// TIA Portal project "StaiteMixare" (V15.1)

(* hardware
DEVICE "S71500/ET200MP station_1"  S7-1500 station
   slot 0: "Rail_0"  Rack  6ES7 590-1***0-0AA0
   slot 1: "PLC_1"  CPU 1513-1 PN  6ES7 513-1AL02-0AB0  V2.6
      slot 3: "CPU display_1"  6ES7591-1AA00-0AA0
DEVICE "HMI_1"  KTP900 Basic PN
   slot 0: "HMI_1"  KTP900 Basic PN  6AV2 123-2JB03-0AX0  15.1.0.0
   slot 1: "HMI_RT_1"  KTP900 Basic PN  6AV2 123-2JB03-0AX0  15.1.0.0
   slot 5: "HMI_1.IE_CP_1"  PROFINET Interface  15.0.1.0
      slot 1: "PROFINET Interface_1"  PROFINET Interface
         slot 1: "Port_1"  Port
*)

// ===== PLC "PLC_1"  CPU 1513-1 PN =====

VAR_GLOBAL   // PLC tag table "Default tag table"
   "Clock_Byte" AT %MB0 : Byte;
   "Clock_10Hz" AT %M0.0 : Bool;
   "Clock_5Hz" AT %M0.1 : Bool;
   "Clock_2.5Hz" AT %M0.2 : Bool;
   "Clock_2Hz" AT %M0.3 : Bool;
   "Clock_1.25Hz" AT %M0.4 : Bool;
   "Clock_1Hz" AT %M0.5 : Bool;
   "Clock_0.625Hz" AT %M0.6 : Bool;
   "Clock_0.5Hz" AT %M0.7 : Bool;
END_VAR

DATA_BLOCK "Alarme"   // DB1
{ S7_Optimized_Access := 'TRUE' }
VERSION : 0.1
   VAR
      alarme_gather : Word;
      alarme_vect : Array[0..15] of Bool;
   END_VAR
BEGIN
END_DATA_BLOCK

DATA_BLOCK "Avarii"   // DB2
{ S7_Optimized_Access := 'TRUE' }
VERSION : 0.1
   VAR
      ESD : Bool;
      esd_btn : Bool;
      reset_esd : Bool;
      avarie_mixer : Bool;
      avarie_container : Bool;
      avarie_solutie_A : Bool;
      avarie_solutie_B : Bool;
      avarie_generala : Bool;
      reset_avarie_generala : Bool;
   END_VAR
BEGIN
END_DATA_BLOCK

DATA_BLOCK "Mixer_DB"   // DB3
{ S7_Optimized_Access := 'TRUE' }
VERSION : 0.1
   VAR
      durata_mixer : Time;
      timp_trecut_secunde : Time;
      timp_elapsed : Time;
      mixer_pornit : Bool;
      plecare_stea : Bool;
      plecare_triunghi : Bool;
      btn_pornire : Bool;
   END_VAR
BEGIN
END_DATA_BLOCK

DATA_BLOCK "Container_DB"   // DB4
{ S7_Optimized_Access := 'TRUE' }
VERSION : 0.1
   VAR
      recipient : Bool := true;
      valva_golire_deschisa : Bool;
      pornire_golire : Bool;
      btn_pornire : Bool;
      debit_total : UInt := 100;
      debit_curent : UInt;
      debit_recipient : UInt := 5;
   END_VAR
BEGIN
END_DATA_BLOCK

DATA_BLOCK "Solutie_A_DB"   // DB5
{ S7_Optimized_Access := 'TRUE' }
VERSION : 0.1
   VAR
      debit_solutie : UInt := 60;
      debit_aux : UInt;
      debit_de_umplut : UInt := 20;
      debit_curent : UInt;
      indice : UInt := 1;
      btn_reumplere : Bool;
      capacitate_necesara : Bool;
      btn_pornire : Bool;
      pornite_golire : Bool;
   END_VAR
BEGIN
END_DATA_BLOCK

DATA_BLOCK "Solutie_B_DB"   // DB6
{ S7_Optimized_Access := 'TRUE' }
VERSION : 0.1
   VAR
      debit_solutie : UInt := 60;
      debit_aux : UInt;
      debit_de_umplut : UInt := 20;
      debit_curent : UInt;
      indice : UInt := 2;
      btn_reumplere : Bool;
      capacitate_necesara : Bool;
      btn_pornire : Bool;
      pornite_golire : Bool;
   END_VAR
BEGIN
END_DATA_BLOCK

DATA_BLOCK "Simulare_DB"   // DB7
{ S7_Optimized_Access := 'TRUE' }
VERSION : 0.1
   VAR
      resetare_proces : Bool;
      terminat_proces : Bool;
      re_stea : Bool;
      re_triunghi : Bool;
      add_stea : UInt;
      add_triunghi : UInt;
      paritate_stea : UInt;
      paritate_triunghi : UInt;
      nume : String;
   END_VAR
BEGIN
END_DATA_BLOCK

DATA_BLOCK "Auxiliare"   // DB8
{ S7_Optimized_Access := 'TRUE' }
VERSION : 0.1
   VAR
      intrece_limita_container : Bool;
      debit_suma : UInt;
   END_VAR
BEGIN
END_DATA_BLOCK

DATA_BLOCK "Butoane/Permisiuni"   // DB11
{ S7_Optimized_Access := 'TRUE' }
VERSION : 0.1
   VAR
      btn_start : Bool;
      permisiune_start : Bool;
      terminat_umplere : Bool;
      terminat_umplere_A : Bool;
      terminat_umplere_B : Bool;
      terminat_golire : Bool;
      terminat_mixer : Bool;
   END_VAR
BEGIN
END_DATA_BLOCK

DATA_BLOCK "Mixer_DB_1"   // DB12
{ S7_Optimized_Access := 'TRUE' }
VERSION : 0.1
// stored: InstanceOfName Mixer
"Mixer"
BEGIN
END_DATA_BLOCK

DATA_BLOCK "Container_DB_1"   // DB13
{ S7_Optimized_Access := 'TRUE' }
VERSION : 0.1
// stored: InstanceOfName Container
"Container"
BEGIN
END_DATA_BLOCK

DATA_BLOCK "SolutieA_DB"   // DB14
{ S7_Optimized_Access := 'TRUE' }
VERSION : 0.1
// stored: InstanceOfName Solutie
"Solutie"
BEGIN
END_DATA_BLOCK

DATA_BLOCK "SolutieB_DB"   // DB15
{ S7_Optimized_Access := 'TRUE' }
VERSION : 0.1
// stored: InstanceOfName Solutie
"Solutie"
BEGIN
END_DATA_BLOCK

DATA_BLOCK "Simulare_DB_1"   // DB16
{ S7_Optimized_Access := 'TRUE' }
VERSION : 0.1
// stored: InstanceOfName Simulare
"Simulare"
BEGIN
END_DATA_BLOCK

DATA_BLOCK "Variabile_HMI"   // DB17
{ S7_Optimized_Access := 'TRUE' }
VERSION : 0.1
   VAR
      stea_1 : Bool;
      stea_2 : Bool;
      triunghi_1 : Bool;
      triunghi_2 : Bool;
   END_VAR
BEGIN
END_DATA_BLOCK

DATA_BLOCK "Date_SCL"   // DB18
{ S7_Optimized_Access := 'TRUE' }
VERSION : 0.1
   VAR
      array_durata : Array[0..99] of Time;
      array_cantitate_A : Array[0..99] of UInt;
      array_cantitate_B : Array[0..99] of UInt;
      array_nume : Array[0..99] of String;
      btn_cauta_nume : Bool;
      btn_cauta_index : Bool;
      btn_salvare : Bool;
      btn_load : Bool;
      index : Int;
      valoare_durata : Time;
      valoare_cantitate_A : UInt;
      valoare_cantitate_B : UInt;
      nume : String;
      index_for : Int;
   END_VAR
BEGIN
END_DATA_BLOCK

// folder: System blocks/Program resources

DATA_BLOCK "Reset_ESD"   // DB9
{ S7_Optimized_Access := 'TRUE' }
AUTHOR : Simatic
FAMILY : IEC
NAME : IEC_TMR
VERSION : 1.0
// stored: InstanceOfName IEC_TIMER
"IEC_TIMER"
BEGIN
END_DATA_BLOCK

DATA_BLOCK "Reset_avarie_generala"   // DB10
{ S7_Optimized_Access := 'TRUE' }
AUTHOR : Simatic
FAMILY : IEC
NAME : IEC_TMR
VERSION : 1.0
// stored: InstanceOfName IEC_TIMER
"IEC_TIMER"
BEGIN
END_DATA_BLOCK

DATA_BLOCK "Resetare_save"   // DB19
{ S7_Optimized_Access := 'TRUE' }
AUTHOR : Simatic
FAMILY : IEC
NAME : IEC_TMR
VERSION : 1.0
// stored: InstanceOfName IEC_TIMER
"IEC_TIMER"
BEGIN
END_DATA_BLOCK

DATA_BLOCK "Resetare_cautare"   // DB20
{ S7_Optimized_Access := 'TRUE' }
AUTHOR : Simatic
FAMILY : IEC
NAME : IEC_TMR
VERSION : 1.0
// stored: InstanceOfName IEC_TIMER
"IEC_TIMER"
BEGIN
END_DATA_BLOCK

DATA_BLOCK "Resetare_load"   // DB21
{ S7_Optimized_Access := 'TRUE' }
AUTHOR : Simatic
FAMILY : IEC
NAME : IEC_TMR
VERSION : 1.0
// stored: InstanceOfName IEC_TIMER
"IEC_TIMER"
BEGIN
END_DATA_BLOCK

DATA_BLOCK "Reset_cautare_index"   // DB22
{ S7_Optimized_Access := 'TRUE' }
AUTHOR : Simatic
FAMILY : IEC
NAME : IEC_TMR
VERSION : 1.0
// stored: InstanceOfName IEC_TIMER
"IEC_TIMER"
BEGIN
END_DATA_BLOCK

// folder: (top level)

FUNCTION_BLOCK "Simulare"   // FB1, LAD
{ S7_Optimized_Access := 'TRUE' }
VERSION : 0.1
   VAR_INPUT
      permisiune_pornire : Bool;
      debit_A : UInt;
      debit_B : UInt;
      debit_cerut_total : UInt;
      terminat_A : Bool;
      terminat_B : Bool;
      terminat_mixer : Bool;
      alarma_A : Bool;
      alarma_B : Bool;
      terminat_golire : Bool;
   END_VAR
   VAR_OUTPUT
      pornire_mixer : Bool;
      pornire_golire : Bool;
      terminat_umplere : Bool;
      terminat_proces : Bool;
      alarma_terminat : Bool;
   END_VAR
   VAR_IN_OUT
      debit_container : UInt;
      plecare_A : Bool;
      plecare_B : Bool;
      resetare_proces : Bool;
   END_VAR
   VAR
      re1 : Bool;
      re2 : Bool;
      timer_resetare : TON_TIME;
   END_VAR
   VAR_TEMP   // added for the SCL form of the ladder/FBD networks
      _w1 : Bool;
      _w2 : Bool;
   END_VAR
BEGIN

REGION Network 1: Permisiune de pornire pe solutia A
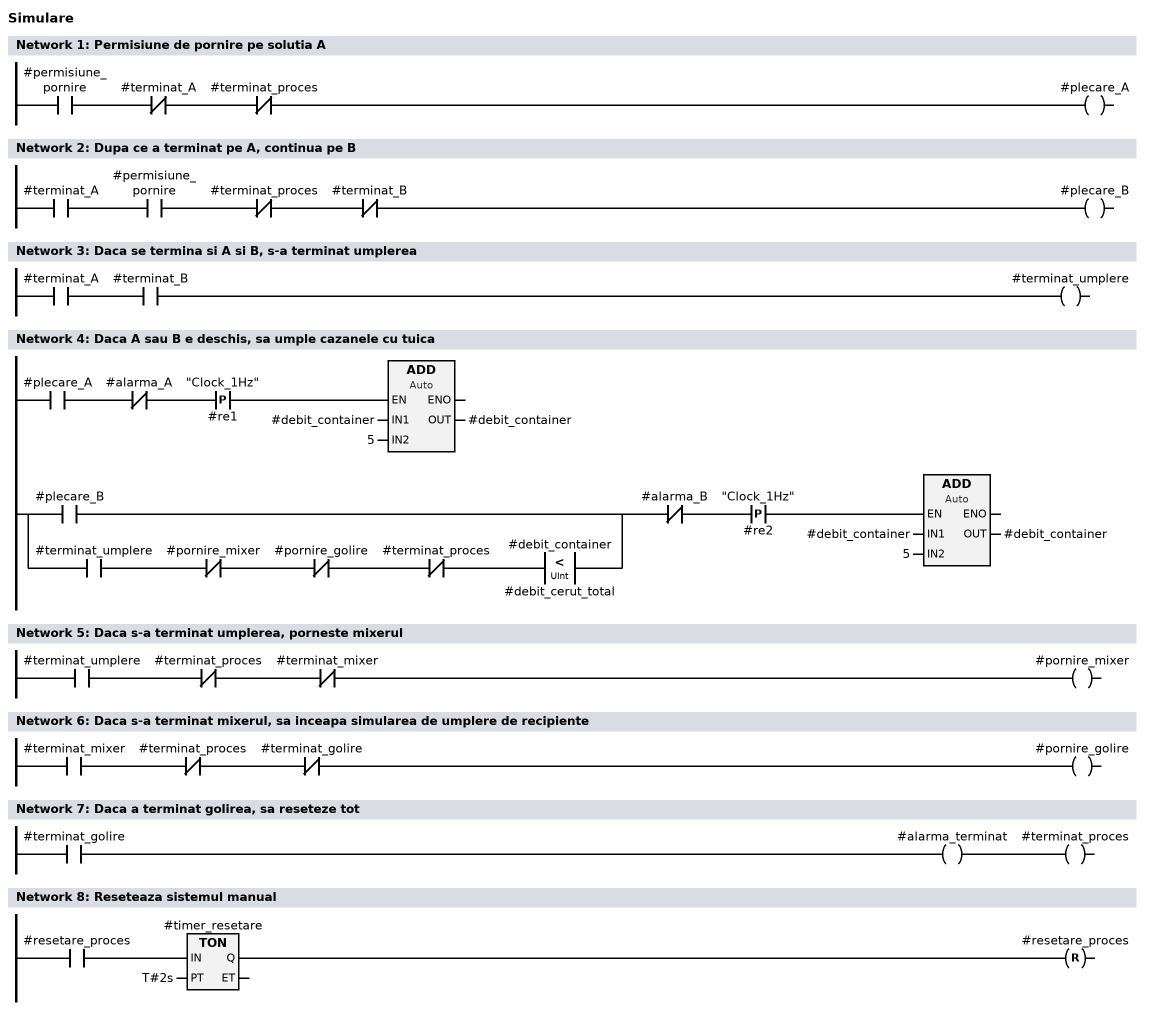
   RUNG wire#powerrail
      Contact( #permisiune_pornire )
      I_Contact( #terminat_A )
      I_Contact( #terminat_proces )
      Coil( #plecare_A )
   END_RUNG
   // the same network as SCL:
   #plecare_A := #permisiune_pornire AND NOT #terminat_A AND NOT #terminat_proces;
END_REGION

REGION Network 2: Dupa ce a terminat pe A, continua pe B
   RUNG wire#powerrail
      Contact( #terminat_A )
      Contact( #permisiune_pornire )
      I_Contact( #terminat_proces )
      I_Contact( #terminat_B )
      Coil( #plecare_B )
   END_RUNG
   // the same network as SCL:
   #plecare_B := #terminat_A AND #permisiune_pornire AND NOT #terminat_proces AND NOT #terminat_B;
END_REGION

REGION Network 3: Daca se termina si A si B, s-a terminat umplerea
   RUNG wire#powerrail
      Contact( #terminat_A )
      Contact( #terminat_B )
      Coil( #terminat_umplere )
   END_RUNG
   // the same network as SCL:
   #terminat_umplere := #terminat_A AND #terminat_B;
END_REGION

REGION Network 4: Daca A sau B e deschis, sa umple cazanele cu tuica
   RUNG wire#powerrail
      Contact( #plecare_A )
      I_Contact( #alarma_A )
      P_Contact(operand := "Clock_1Hz", bit := #re1)
      Add(in1 := #debit_container, in2 := 5, out => #debit_container)
   END_RUNG
   RUNG wire#powerrail
      Contact( #plecare_B )
      wire#w1
      I_Contact( #alarma_B )
      P_Contact(operand := "Clock_1Hz", bit := #re2)
      Add(in1 := #debit_container, in2 := 5, out => #debit_container)
   END_RUNG
   RUNG wire#powerrail
      Contact( #terminat_umplere )
      I_Contact( #pornire_mixer )
      I_Contact( #pornire_golire )
      I_Contact( #terminat_proces )
      { S7_Templates := "SrcType := UInt" } LT_Contact(in1 := #debit_container, in2 := #debit_cerut_total)
   END_RUNG wire#w1
   // the same network as SCL:
   #_w1 := #plecare_A AND NOT #alarma_A AND "Clock_1Hz" AND NOT #re1;   // rising edge of "Clock_1Hz"
   #re1 := "Clock_1Hz";
   IF #_w1 THEN #debit_container := #debit_container + 5; END_IF;
   #_w2 := (#plecare_B OR (#terminat_umplere AND NOT #pornire_mixer AND NOT #pornire_golire AND NOT #terminat_proces AND (#debit_container < #debit_cerut_total))) AND NOT #alarma_B AND "Clock_1Hz" AND NOT #re2;   // rising edge of "Clock_1Hz"
   #re2 := "Clock_1Hz";
   IF #_w2 THEN #debit_container := #debit_container + 5; END_IF;
END_REGION

REGION Network 5: Daca s-a terminat umplerea, porneste mixerul
   RUNG wire#powerrail
      Contact( #terminat_umplere )
      I_Contact( #terminat_proces )
      I_Contact( #terminat_mixer )
      Coil( #pornire_mixer )
   END_RUNG
   // the same network as SCL:
   #pornire_mixer := #terminat_umplere AND NOT #terminat_proces AND NOT #terminat_mixer;
END_REGION

REGION Network 6: Daca s-a terminat mixerul, sa inceapa simularea de umplere de recipiente
   RUNG wire#powerrail
      Contact( #terminat_mixer )
      I_Contact( #terminat_proces )
      I_Contact( #terminat_golire )
      Coil( #pornire_golire )
   END_RUNG
   // the same network as SCL:
   #pornire_golire := #terminat_mixer AND NOT #terminat_proces AND NOT #terminat_golire;
END_REGION

REGION Network 7: Daca a terminat golirea, sa reseteze tot
   RUNG wire#powerrail
      Contact( #terminat_golire )
      Coil( #alarma_terminat )
      Coil( #terminat_proces )
   END_RUNG
   // the same network as SCL:
   #alarma_terminat := #terminat_golire;
   #terminat_proces := #terminat_golire;
END_REGION

REGION Network 8: Reseteaza sistemul manual
   #timer_resetare(IN := #resetare_proces, PT := T#2s);   // TON
   IF #timer_resetare.Q THEN #resetare_proces := FALSE; END_IF;
END_REGION
END_FUNCTION_BLOCK

FUNCTION_BLOCK "Container"   // FB2, LAD
{ S7_Optimized_Access := 'TRUE' }
VERSION : 0.1
   VAR_INPUT
      esd : Bool;
      avarie_generala : Bool;
      terminat_mixer : Bool;
      resetare_sistem : Bool;
      permisiune_pornire : Bool;
   END_VAR
   VAR_OUTPUT
      pornire_golire : Bool;
      valva_golire_deschisa : Bool;
      terminat_golire : Bool;
   END_VAR
   VAR_IN_OUT
      recipient : Bool;
      debit_total : UInt;
      debit_recipient : UInt;
      debit_curent : UInt;
      btn_pornire : Bool;
   END_VAR
   VAR
      re1 : Bool;
      debit_aux : UInt;
      container_gol : Bool;
      timer_recipient : TON_TIME;
   END_VAR
   VAR_TEMP   // added for the SCL form of the ladder/FBD networks
      _w1 : Bool;
   END_VAR
BEGIN

REGION Network 1: Conditie pornire
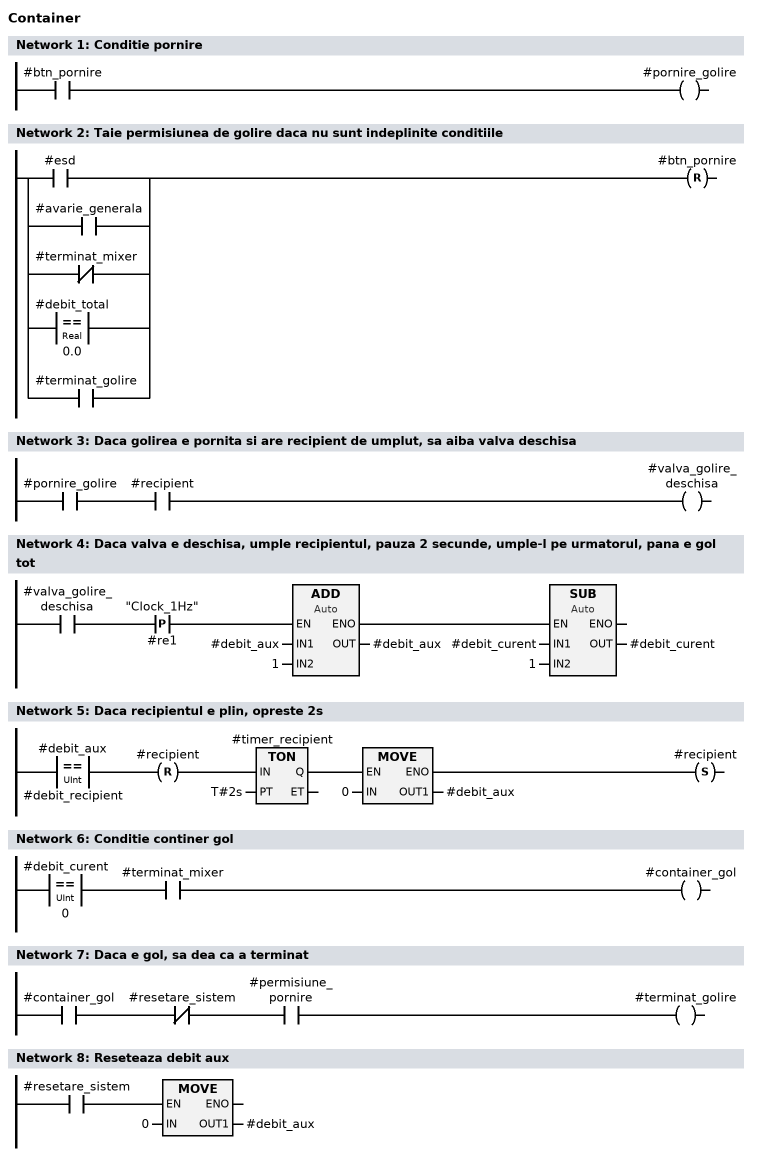
   RUNG wire#powerrail
      Contact( #btn_pornire )
      Coil( #pornire_golire )
   END_RUNG
   // the same network as SCL:
   #pornire_golire := #btn_pornire;
END_REGION

REGION Network 2: Taie permisiunea de golire daca nu sunt indeplinite conditiile
   RUNG wire#powerrail
      Contact( #esd )
      wire#w1
      R_Coil( #btn_pornire )
   END_RUNG
   RUNG wire#powerrail
      Contact( #avarie_generala )
   END_RUNG wire#w1
   RUNG wire#powerrail
      I_Contact( #terminat_mixer )
   END_RUNG wire#w1
   RUNG wire#powerrail
      { S7_Templates := "SrcType := Real" } EQ_Contact(in1 := #debit_total, in2 := 0.0)
   END_RUNG wire#w1
   RUNG wire#powerrail
      Contact( #terminat_golire )
   END_RUNG wire#w1
   // the same network as SCL:
   IF #esd OR #avarie_generala OR NOT #terminat_mixer OR (#debit_total = 0.0) OR #terminat_golire THEN
       #btn_pornire := FALSE;
   END_IF;
END_REGION

REGION Network 3: Daca golirea e pornita si are recipient de umplut, sa aiba valva deschisa
   RUNG wire#powerrail
      Contact( #pornire_golire )
      Contact( #recipient )
      Coil( #valva_golire_deschisa )
   END_RUNG
   // the same network as SCL:
   #valva_golire_deschisa := #pornire_golire AND #recipient;
END_REGION

REGION Network 4: Daca valva e deschisa, umple recipientul, pauza 2 secunde, umple-l pe urmatorul, pana e gol tot
   RUNG wire#powerrail
      Contact( #valva_golire_deschisa )
      P_Contact(operand := "Clock_1Hz", bit := #re1)
      Add(in1 := #debit_aux, in2 := 1, out => #debit_aux)
      Sub(in1 := #debit_curent, in2 := 1, out => #debit_curent)
   END_RUNG
   // the same network as SCL:
   #_w1 := #valva_golire_deschisa AND "Clock_1Hz" AND NOT #re1;   // rising edge of "Clock_1Hz"
   #re1 := "Clock_1Hz";
   IF #_w1 THEN
       #debit_aux := #debit_aux + 1;
       #debit_curent := #debit_curent - 1;
   END_IF;
END_REGION

REGION Network 5: Daca recipientul e plin, opreste 2s
   #_w1 := #debit_aux = #debit_recipient;
   IF #_w1 THEN #recipient := FALSE; END_IF;
   #timer_recipient(IN := #_w1, PT := T#2s);   // TON
   IF #timer_recipient.Q THEN
       #debit_aux := 0;
       #recipient := TRUE;
   END_IF;
END_REGION

REGION Network 6: Conditie continer gol
   RUNG wire#powerrail
      { S7_Templates := "SrcType := UInt" } EQ_Contact(in1 := #debit_curent, in2 := 0)
      Contact( #terminat_mixer )
      Coil( #container_gol )
   END_RUNG
   // the same network as SCL:
   #container_gol := (#debit_curent = 0) AND #terminat_mixer;
END_REGION

REGION Network 7: Daca e gol, sa dea ca a terminat
   RUNG wire#powerrail
      Contact( #container_gol )
      I_Contact( #resetare_sistem )
      Contact( #permisiune_pornire )
      Coil( #terminat_golire )
   END_RUNG
   // the same network as SCL:
   #terminat_golire := #container_gol AND NOT #resetare_sistem AND #permisiune_pornire;
END_REGION

REGION Network 8: Reseteaza debit aux
   RUNG wire#powerrail
      Contact( #resetare_sistem )
      Move(in := 0, out1 => #debit_aux)
   END_RUNG
   // the same network as SCL:
   IF #resetare_sistem THEN #debit_aux := 0; END_IF;
END_REGION
END_FUNCTION_BLOCK

FUNCTION_BLOCK "Solutie"   // FB3, LAD
{ S7_Optimized_Access := 'TRUE' }
VERSION : 0.1
   VAR_INPUT
      esd : Bool;
      avarie : Bool;
      debit_solutie : UInt;
      debit_cerut : UInt;
      resetare_sistem : Bool;
   END_VAR
   VAR_OUTPUT
      debit_curent : UInt;
      alarma : Bool;
      pornire_golire : Bool;
   END_VAR
   VAR_IN_OUT
      debit_aux : UInt;
      btn_reumplere_solutie : Bool;
      capacitate_necesara : Bool;
      btn_pornire : Bool;
      terminat_umplere : Bool;
   END_VAR
   VAR
      re1 : Bool;
      timer_reset_btn_reumplere : TON_TIME;
   END_VAR
   VAR_TEMP   // added for the SCL form of the ladder/FBD networks
      _w1 : Bool;
      _w2 : Bool;
   END_VAR
BEGIN

REGION Network 1: Calcul daca are suficienta solutie
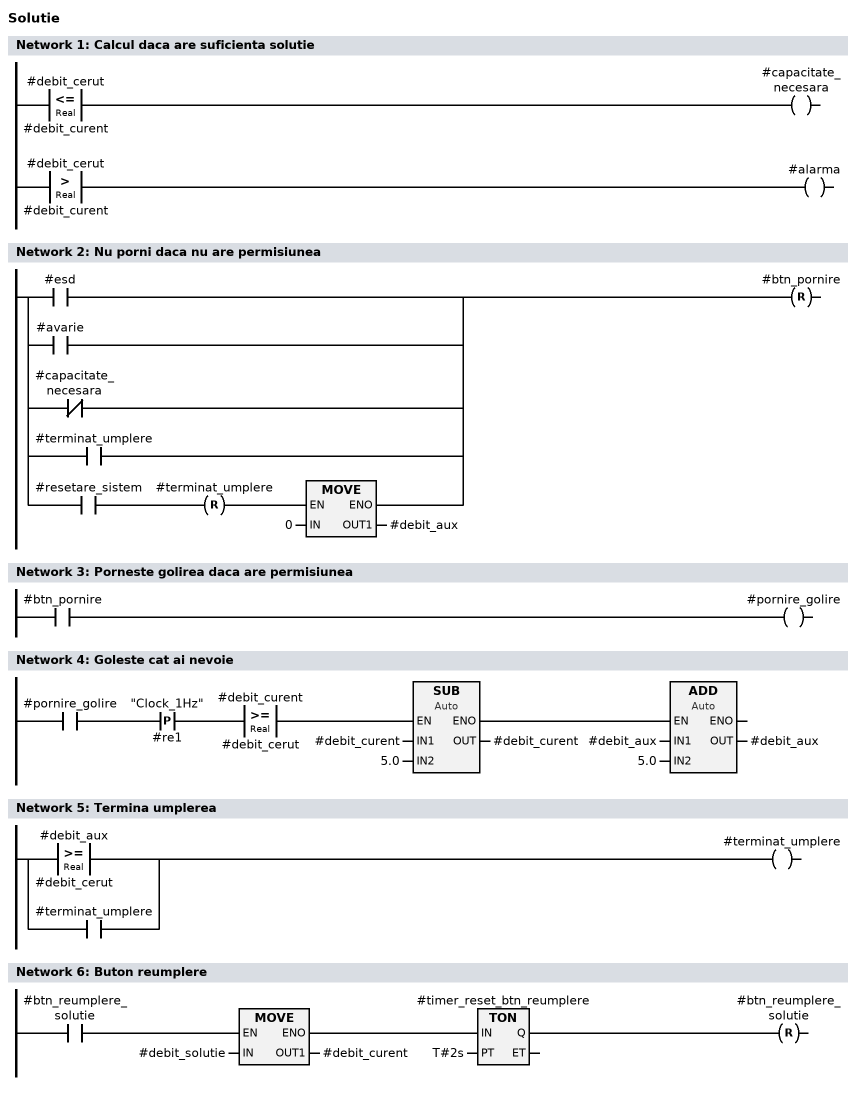
   RUNG wire#powerrail
      { S7_Templates := "SrcType := Real" } LE_Contact(in1 := #debit_cerut, in2 := #debit_curent)
      Coil( #capacitate_necesara )
   END_RUNG
   RUNG wire#powerrail
      { S7_Templates := "SrcType := Real" } GT_Contact(in1 := #debit_cerut, in2 := #debit_curent)
      Coil( #alarma )
   END_RUNG
   // the same network as SCL:
   #capacitate_necesara := #debit_cerut <= #debit_curent;
   #alarma := #debit_cerut > #debit_curent;
END_REGION

REGION Network 2: Nu porni daca nu are permisiunea
   RUNG wire#powerrail
      Contact( #esd )
      wire#w1
      R_Coil( #btn_pornire )
   END_RUNG
   RUNG wire#powerrail
      Contact( #avarie )
   END_RUNG wire#w1
   RUNG wire#powerrail
      I_Contact( #capacitate_necesara )
   END_RUNG wire#w1
   RUNG wire#powerrail
      Contact( #terminat_umplere )
   END_RUNG wire#w1
   RUNG wire#powerrail
      Contact( #resetare_sistem )
      R_Coil( #terminat_umplere )
      Move(in := 0, out1 => #debit_aux)
   END_RUNG wire#w1
   // the same network as SCL:
   #_w1 := #terminat_umplere;
   IF #resetare_sistem THEN
       #terminat_umplere := FALSE;
       #debit_aux := 0;
   END_IF;
   IF #esd OR #avarie OR NOT #capacitate_necesara OR #_w1 OR #resetare_sistem THEN
       #btn_pornire := FALSE;
   END_IF;
END_REGION

REGION Network 3: Porneste golirea daca are permisiunea
   RUNG wire#powerrail
      Contact( #btn_pornire )
      Coil( #pornire_golire )
   END_RUNG
   // the same network as SCL:
   #pornire_golire := #btn_pornire;
END_REGION

REGION Network 4: Goleste cat ai nevoie
   RUNG wire#powerrail
      Contact( #pornire_golire )
      P_Contact(operand := "Clock_1Hz", bit := #re1)
      { S7_Templates := "SrcType := Real" } GE_Contact(in1 := #debit_curent, in2 := #debit_cerut)
      Sub(in1 := #debit_curent, in2 := 5.0, out => #debit_curent)
      Add(in1 := #debit_aux, in2 := 5.0, out => #debit_aux)
   END_RUNG
   // the same network as SCL:
   #_w1 := #pornire_golire AND "Clock_1Hz" AND NOT #re1;   // rising edge of "Clock_1Hz"
   #re1 := "Clock_1Hz";
   #_w2 := #_w1 AND (#debit_curent >= #debit_cerut);
   IF #_w2 THEN
       #debit_curent := #debit_curent - 5.0;
       #debit_aux := #debit_aux + 5.0;
   END_IF;
END_REGION

REGION Network 5: Termina umplerea
   RUNG wire#powerrail
      { S7_Templates := "SrcType := Real" } GE_Contact(in1 := #debit_aux, in2 := #debit_cerut)
      wire#w1
      Coil( #terminat_umplere )
   END_RUNG
   RUNG wire#powerrail
      Contact( #terminat_umplere )
   END_RUNG wire#w1
   // the same network as SCL:
   #terminat_umplere := (#debit_aux >= #debit_cerut) OR #terminat_umplere;
END_REGION

REGION Network 6: Buton reumplere
   IF #btn_reumplere_solutie THEN #debit_curent := #debit_solutie; END_IF;
   #timer_reset_btn_reumplere(IN := #btn_reumplere_solutie, PT := T#2s);   // TON
   IF #timer_reset_btn_reumplere.Q THEN #btn_reumplere_solutie := FALSE; END_IF;
END_REGION
END_FUNCTION_BLOCK

FUNCTION_BLOCK "Mixer"   // FB4, LAD
{ S7_Optimized_Access := 'TRUE' }
VERSION : 0.1
   VAR_INPUT
      esd : Bool;
      avarie_generala : Bool;
      terminat_umplere : Bool;
      durata_mixer : Time;
      resetare_proces : Bool;
   END_VAR
   VAR_OUTPUT
      mixer_pornit : Bool;
      timp_triunghi_secunde : Time;
      terminat_mixer : Bool;
      timp_trecut : Time;
   END_VAR
   VAR_IN_OUT
      plecare_stea : Bool;
      plecare_triunghi : Bool;
      btn_pornire : Bool;
   END_VAR
   VAR
      timer_stea : TON_TIME;
      timp_trecut_ms : Time;
      timer_triunghi : TON_TIME;
   END_VAR
   VAR_TEMP   // added for the SCL form of the ladder/FBD networks
      _w1 : Bool;
   END_VAR
BEGIN

REGION Network 1: Conditie de pornire (stea)
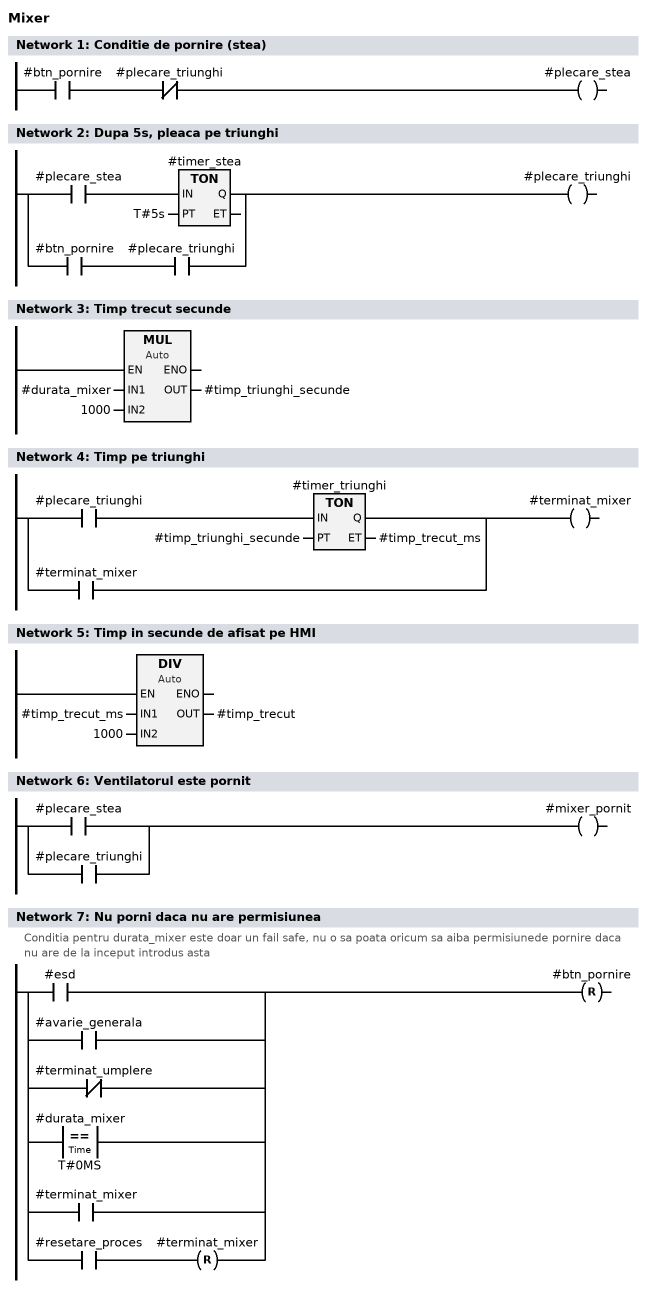
   RUNG wire#powerrail
      Contact( #btn_pornire )
      I_Contact( #plecare_triunghi )
      Coil( #plecare_stea )
   END_RUNG
   // the same network as SCL:
   #plecare_stea := #btn_pornire AND NOT #plecare_triunghi;
END_REGION

REGION Network 2: Dupa 5s, pleaca pe triunghi
   #timer_stea(IN := #plecare_stea, PT := T#5s);   // TON
   #plecare_triunghi := #timer_stea.Q OR (#btn_pornire AND #plecare_triunghi);
END_REGION

REGION Network 3: Timp trecut secunde
   RUNG wire#powerrail
      Mul(in1 := #durata_mixer, in2 := 1000, out => #timp_triunghi_secunde)
   END_RUNG
   // the same network as SCL:
   #timp_triunghi_secunde := #durata_mixer * 1000;
END_REGION

REGION Network 4: Timp pe triunghi
   #timer_triunghi(IN := #plecare_triunghi, PT := #timp_triunghi_secunde, ET => #timp_trecut_ms);   // TON
   #terminat_mixer := #timer_triunghi.Q OR #terminat_mixer;
END_REGION

REGION Network 5: Timp in secunde de afisat pe HMI
   RUNG wire#powerrail
      Div(in1 := #timp_trecut_ms, in2 := 1000, out => #timp_trecut)
   END_RUNG
   // the same network as SCL:
   #timp_trecut := #timp_trecut_ms / 1000;
END_REGION

REGION Network 6: Ventilatorul este pornit
   RUNG wire#powerrail
      Contact( #plecare_stea )
      wire#w1
      Coil( #mixer_pornit )
   END_RUNG
   RUNG wire#powerrail
      Contact( #plecare_triunghi )
   END_RUNG wire#w1
   // the same network as SCL:
   #mixer_pornit := #plecare_stea OR #plecare_triunghi;
END_REGION

REGION Network 7: Nu porni daca nu are permisiunea
   // Conditia pentru durata_mixer este doar un fail safe, nu o sa poata oricum sa aiba permisiunede pornire daca nu are de la inceput introdus asta
   RUNG wire#powerrail
      Contact( #esd )
      wire#w1
      R_Coil( #btn_pornire )
   END_RUNG
   RUNG wire#powerrail
      Contact( #avarie_generala )
   END_RUNG wire#w1
   RUNG wire#powerrail
      I_Contact( #terminat_umplere )
   END_RUNG wire#w1
   RUNG wire#powerrail
      { S7_Templates := "SrcType := Time" } EQ_Contact(in1 := #durata_mixer, in2 := T#0MS)
   END_RUNG wire#w1
   RUNG wire#powerrail
      Contact( #terminat_mixer )
   END_RUNG wire#w1
   RUNG wire#powerrail
      Contact( #resetare_proces )
      R_Coil( #terminat_mixer )
   END_RUNG wire#w1
   // the same network as SCL:
   #_w1 := #terminat_mixer;
   IF #resetare_proces THEN #terminat_mixer := FALSE; END_IF;
   IF #esd OR #avarie_generala OR NOT #terminat_umplere OR (#durata_mixer = T#0MS) OR #_w1 OR #resetare_proces THEN
       #btn_pornire := FALSE;
   END_IF;
END_REGION
END_FUNCTION_BLOCK

ORGANIZATION_BLOCK "Main"   // OB1, LAD, ProgramCycle
TITLE = "Main Program Sweep (Cycle)"
{ S7_Optimized_Access := 'TRUE' }
VERSION : 0.1
   VAR_INPUT
      Initial_Call : Bool;   // Initial call of this OB
      Remanence : Bool;   // =True, if remanent data are available
   END_VAR
   VAR_TEMP   // added for the SCL form of the ladder/FBD networks
      _w1 : Bool;
      _w2 : Bool;
   END_VAR
BEGIN

REGION Network 1: Gather pe alarme
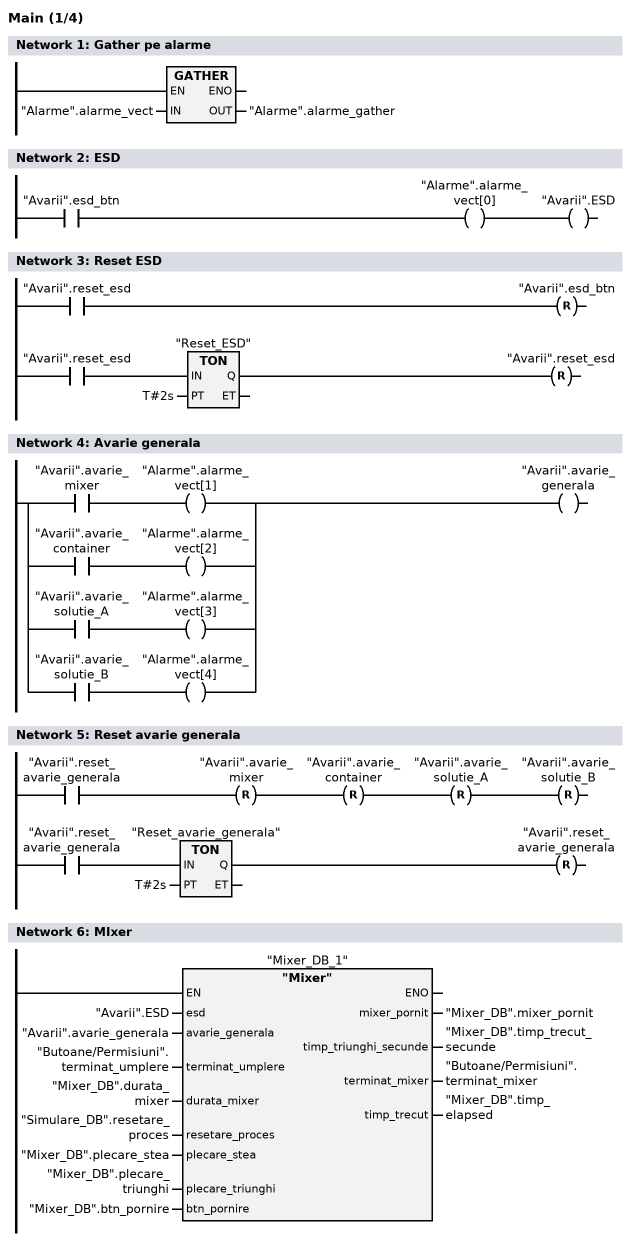
   GATHER(IN := "Alarme".alarme_vect, OUT => "Alarme".alarme_gather);
END_REGION

REGION Network 2: ESD
   RUNG wire#powerrail
      Contact( "Avarii".esd_btn )
      Coil( "Alarme".alarme_vect[0] )
      Coil( "Avarii".ESD )
   END_RUNG
   // the same network as SCL:
   "Alarme".alarme_vect[0] := "Avarii".esd_btn;
   "Avarii".ESD := "Avarii".esd_btn;
END_REGION

REGION Network 3: Reset ESD
   IF "Avarii".reset_esd THEN "Avarii".esd_btn := FALSE; END_IF;
   "Reset_ESD".TON(IN := "Avarii".reset_esd, PT := T#2s);
   IF "Reset_ESD".Q THEN "Avarii".reset_esd := FALSE; END_IF;
END_REGION

REGION Network 4: Avarie generala
   RUNG wire#powerrail
      Contact( "Avarii".avarie_mixer )
      Coil( "Alarme".alarme_vect[1] )
      wire#w1
      Coil( "Avarii".avarie_generala )
   END_RUNG
   RUNG wire#powerrail
      Contact( "Avarii".avarie_container )
      Coil( "Alarme".alarme_vect[2] )
   END_RUNG wire#w1
   RUNG wire#powerrail
      Contact( "Avarii".avarie_solutie_A )
      Coil( "Alarme".alarme_vect[3] )
   END_RUNG wire#w1
   RUNG wire#powerrail
      Contact( "Avarii".avarie_solutie_B )
      Coil( "Alarme".alarme_vect[4] )
   END_RUNG wire#w1
   // the same network as SCL:
   "Alarme".alarme_vect[1] := "Avarii".avarie_mixer;
   "Alarme".alarme_vect[2] := "Avarii".avarie_container;
   "Alarme".alarme_vect[3] := "Avarii".avarie_solutie_A;
   "Alarme".alarme_vect[4] := "Avarii".avarie_solutie_B;
   "Avarii".avarie_generala := "Avarii".avarie_mixer OR "Avarii".avarie_container OR "Avarii".avarie_solutie_A OR "Avarii".avarie_solutie_B;
END_REGION

REGION Network 5: Reset avarie generala
   IF "Avarii".reset_avarie_generala THEN
       "Avarii".avarie_mixer := FALSE;
       "Avarii".avarie_container := FALSE;
       "Avarii".avarie_solutie_A := FALSE;
       "Avarii".avarie_solutie_B := FALSE;
   END_IF;
   "Reset_avarie_generala".TON(IN := "Avarii".reset_avarie_generala, PT := T#2s);
   IF "Reset_avarie_generala".Q THEN "Avarii".reset_avarie_generala := FALSE; END_IF;
END_REGION

REGION Network 6: MIxer
   RUNG wire#powerrail
      "Mixer_DB_1"(esd := "Avarii".ESD, avarie_generala := "Avarii".avarie_generala, terminat_umplere := "Butoane/Permisiuni".terminat_umplere, durata_mixer := "Mixer_DB".durata_mixer, resetare_proces := "Simulare_DB".resetare_proces, plecare_stea := "Mixer_DB".plecare_stea, plecare_triunghi := "Mixer_DB".plecare_triunghi, btn_pornire := "Mixer_DB".btn_pornire, mixer_pornit => "Mixer_DB".mixer_pornit, timp_triunghi_secunde => "Mixer_DB".timp_trecut_secunde, terminat_mixer => "Butoane/Permisiuni".terminat_mixer, timp_trecut => "Mixer_DB".timp_elapsed)
   END_RUNG
   // the same network as SCL:
   "Mixer_DB_1"(esd := "Avarii".ESD,   // "Mixer"
                avarie_generala := "Avarii".avarie_generala,
                terminat_umplere := "Butoane/Permisiuni".terminat_umplere,
                durata_mixer := "Mixer_DB".durata_mixer,
                resetare_proces := "Simulare_DB".resetare_proces,
                plecare_stea := "Mixer_DB".plecare_stea,
                plecare_triunghi := "Mixer_DB".plecare_triunghi,
                btn_pornire := "Mixer_DB".btn_pornire,
                mixer_pornit => "Mixer_DB".mixer_pornit,
                timp_triunghi_secunde => "Mixer_DB".timp_trecut_secunde,
                terminat_mixer => "Butoane/Permisiuni".terminat_mixer,
                timp_trecut => "Mixer_DB".timp_elapsed);
END_REGION

REGION Network 7: HMI motor stea
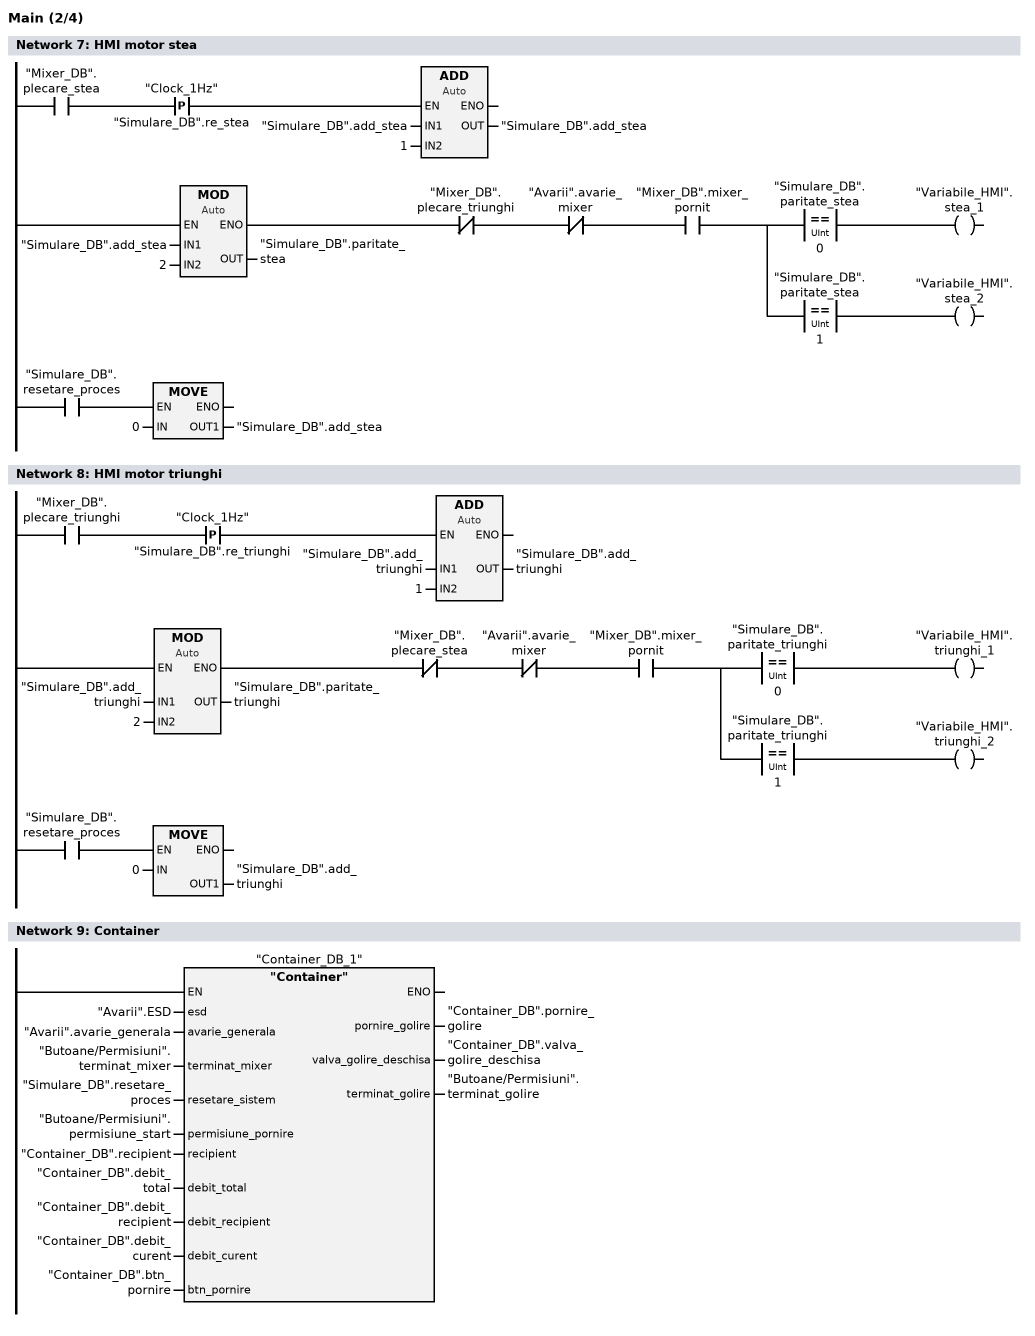
   RUNG wire#powerrail
      Contact( "Mixer_DB".plecare_stea )
      P_Contact(operand := "Clock_1Hz", bit := "Simulare_DB".re_stea)
      Add(in1 := "Simulare_DB".add_stea, in2 := 1, out => "Simulare_DB".add_stea)
   END_RUNG
   RUNG wire#powerrail
      Mod(in1 := "Simulare_DB".add_stea, in2 := 2, out => "Simulare_DB".paritate_stea)
      I_Contact( "Mixer_DB".plecare_triunghi )
      I_Contact( "Avarii".avarie_mixer )
      Contact( "Mixer_DB".mixer_pornit )
      wire#w1
      { S7_Templates := "SrcType := UInt" } EQ_Contact(in1 := "Simulare_DB".paritate_stea, in2 := 0)
      Coil( "Variabile_HMI".stea_1 )
   END_RUNG
   RUNG wire#w1
      { S7_Templates := "SrcType := UInt" } EQ_Contact(in1 := "Simulare_DB".paritate_stea, in2 := 1)
      Coil( "Variabile_HMI".stea_2 )
   END_RUNG
   RUNG wire#powerrail
      Contact( "Simulare_DB".resetare_proces )
      Move(in := 0, out1 => "Simulare_DB".add_stea)
   END_RUNG
   // the same network as SCL:
   #_w1 := "Mixer_DB".plecare_stea AND "Clock_1Hz" AND NOT "Simulare_DB".re_stea;   // rising edge of "Clock_1Hz"
   "Simulare_DB".re_stea := "Clock_1Hz";
   IF #_w1 THEN "Simulare_DB".add_stea := "Simulare_DB".add_stea + 1; END_IF;
   "Simulare_DB".paritate_stea := "Simulare_DB".add_stea MOD 2;
   #_w2 := NOT "Mixer_DB".plecare_triunghi AND NOT "Avarii".avarie_mixer AND "Mixer_DB".mixer_pornit;
   "Variabile_HMI".stea_1 := #_w2 AND ("Simulare_DB".paritate_stea = 0);
   "Variabile_HMI".stea_2 := #_w2 AND ("Simulare_DB".paritate_stea = 1);
   IF "Simulare_DB".resetare_proces THEN "Simulare_DB".add_stea := 0; END_IF;
END_REGION

REGION Network 8: HMI motor triunghi
   RUNG wire#powerrail
      Contact( "Mixer_DB".plecare_triunghi )
      P_Contact(operand := "Clock_1Hz", bit := "Simulare_DB".re_triunghi)
      Add(in1 := "Simulare_DB".add_triunghi, in2 := 1, out => "Simulare_DB".add_triunghi)
   END_RUNG
   RUNG wire#powerrail
      Mod(in1 := "Simulare_DB".add_triunghi, in2 := 2, out => "Simulare_DB".paritate_triunghi)
      I_Contact( "Mixer_DB".plecare_stea )
      I_Contact( "Avarii".avarie_mixer )
      Contact( "Mixer_DB".mixer_pornit )
      wire#w1
      { S7_Templates := "SrcType := UInt" } EQ_Contact(in1 := "Simulare_DB".paritate_triunghi, in2 := 0)
      Coil( "Variabile_HMI".triunghi_1 )
   END_RUNG
   RUNG wire#w1
      { S7_Templates := "SrcType := UInt" } EQ_Contact(in1 := "Simulare_DB".paritate_triunghi, in2 := 1)
      Coil( "Variabile_HMI".triunghi_2 )
   END_RUNG
   RUNG wire#powerrail
      Contact( "Simulare_DB".resetare_proces )
      Move(in := 0, out1 => "Simulare_DB".add_triunghi)
   END_RUNG
   // the same network as SCL:
   #_w1 := "Mixer_DB".plecare_triunghi AND "Clock_1Hz" AND NOT "Simulare_DB".re_triunghi;   // rising edge of "Clock_1Hz"
   "Simulare_DB".re_triunghi := "Clock_1Hz";
   IF #_w1 THEN "Simulare_DB".add_triunghi := "Simulare_DB".add_triunghi + 1; END_IF;
   "Simulare_DB".paritate_triunghi := "Simulare_DB".add_triunghi MOD 2;
   #_w2 := NOT "Mixer_DB".plecare_stea AND NOT "Avarii".avarie_mixer AND "Mixer_DB".mixer_pornit;
   "Variabile_HMI".triunghi_1 := #_w2 AND ("Simulare_DB".paritate_triunghi = 0);
   "Variabile_HMI".triunghi_2 := #_w2 AND ("Simulare_DB".paritate_triunghi = 1);
   IF "Simulare_DB".resetare_proces THEN "Simulare_DB".add_triunghi := 0; END_IF;
END_REGION

REGION Network 9: Container
   RUNG wire#powerrail
      "Container_DB_1"(esd := "Avarii".ESD, avarie_generala := "Avarii".avarie_generala, terminat_mixer := "Butoane/Permisiuni".terminat_mixer, resetare_sistem := "Simulare_DB".resetare_proces, permisiune_pornire := "Butoane/Permisiuni".permisiune_start, recipient := "Container_DB".recipient, debit_total := "Container_DB".debit_total, debit_recipient := "Container_DB".debit_recipient, debit_curent := "Container_DB".debit_curent, btn_pornire := "Container_DB".btn_pornire, pornire_golire => "Container_DB".pornire_golire, valva_golire_deschisa => "Container_DB".valva_golire_deschisa, terminat_golire => "Butoane/Permisiuni".terminat_golire)
   END_RUNG
   // the same network as SCL:
   "Container_DB_1"(esd := "Avarii".ESD,   // "Container"
                    avarie_generala := "Avarii".avarie_generala,
                    terminat_mixer := "Butoane/Permisiuni".terminat_mixer,
                    resetare_sistem := "Simulare_DB".resetare_proces,
                    permisiune_pornire := "Butoane/Permisiuni".permisiune_start,
                    recipient := "Container_DB".recipient,
                    debit_total := "Container_DB".debit_total,
                    debit_recipient := "Container_DB".debit_recipient,
                    debit_curent := "Container_DB".debit_curent,
                    btn_pornire := "Container_DB".btn_pornire,
                    pornire_golire => "Container_DB".pornire_golire,
                    valva_golire_deschisa => "Container_DB".valva_golire_deschisa,
                    terminat_golire => "Butoane/Permisiuni".terminat_golire);
END_REGION

REGION Network 10: Solutie A/B
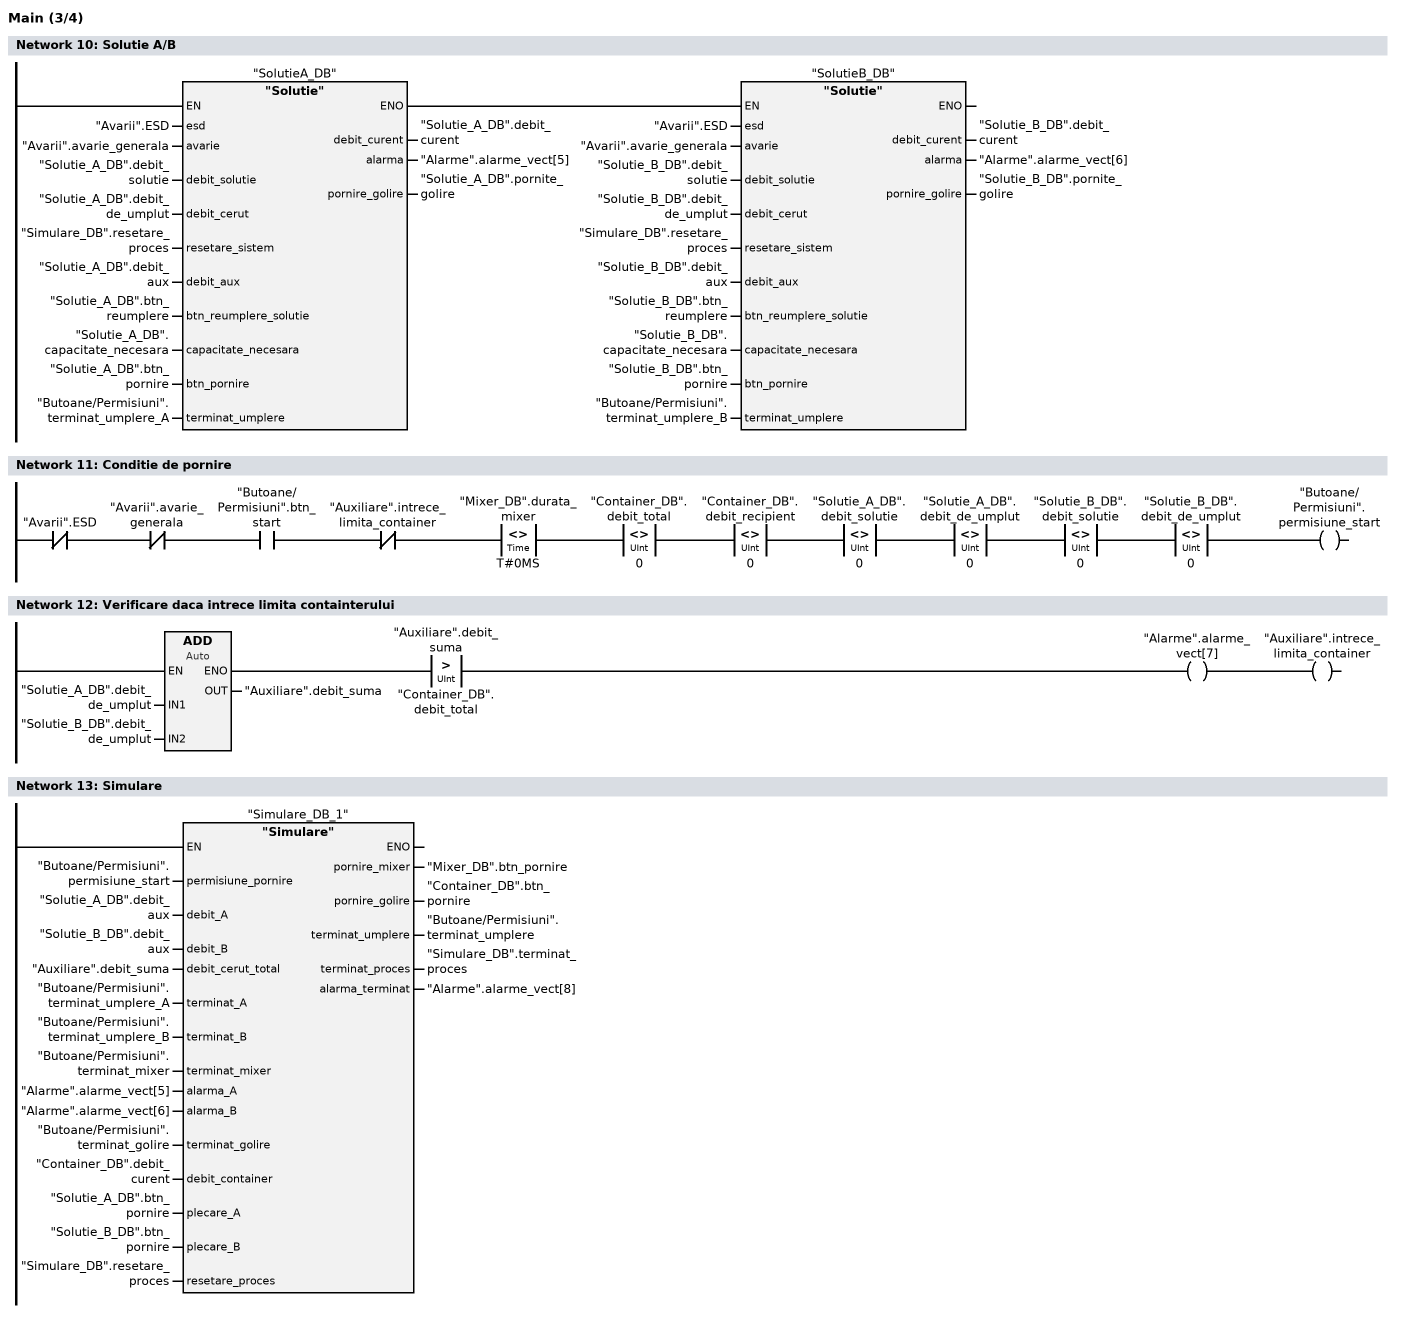
   RUNG wire#powerrail
      "SolutieA_DB"(esd := "Avarii".ESD, avarie := "Avarii".avarie_generala, debit_solutie := "Solutie_A_DB".debit_solutie, debit_cerut := "Solutie_A_DB".debit_de_umplut, resetare_sistem := "Simulare_DB".resetare_proces, debit_aux := "Solutie_A_DB".debit_aux, btn_reumplere_solutie := "Solutie_A_DB".btn_reumplere, capacitate_necesara := "Solutie_A_DB".capacitate_necesara, btn_pornire := "Solutie_A_DB".btn_pornire, terminat_umplere := "Butoane/Permisiuni".terminat_umplere_A, debit_curent => "Solutie_A_DB".debit_curent, alarma => "Alarme".alarme_vect[5], pornire_golire => "Solutie_A_DB".pornite_golire)
      "SolutieB_DB"(esd := "Avarii".ESD, avarie := "Avarii".avarie_generala, debit_solutie := "Solutie_B_DB".debit_solutie, debit_cerut := "Solutie_B_DB".debit_de_umplut, resetare_sistem := "Simulare_DB".resetare_proces, debit_aux := "Solutie_B_DB".debit_aux, btn_reumplere_solutie := "Solutie_B_DB".btn_reumplere, capacitate_necesara := "Solutie_B_DB".capacitate_necesara, btn_pornire := "Solutie_B_DB".btn_pornire, terminat_umplere := "Butoane/Permisiuni".terminat_umplere_B, debit_curent => "Solutie_B_DB".debit_curent, alarma => "Alarme".alarme_vect[6], pornire_golire => "Solutie_B_DB".pornite_golire)
   END_RUNG
   // the same network as SCL:
   "SolutieA_DB"(esd := "Avarii".ESD,   // "Solutie"
                 avarie := "Avarii".avarie_generala,
                 debit_solutie := "Solutie_A_DB".debit_solutie,
                 debit_cerut := "Solutie_A_DB".debit_de_umplut,
                 resetare_sistem := "Simulare_DB".resetare_proces,
                 debit_aux := "Solutie_A_DB".debit_aux,
                 btn_reumplere_solutie := "Solutie_A_DB".btn_reumplere,
                 capacitate_necesara := "Solutie_A_DB".capacitate_necesara,
                 btn_pornire := "Solutie_A_DB".btn_pornire,
                 terminat_umplere := "Butoane/Permisiuni".terminat_umplere_A,
                 debit_curent => "Solutie_A_DB".debit_curent,
                 alarma => "Alarme".alarme_vect[5],
                 pornire_golire => "Solutie_A_DB".pornite_golire,
                 ENO => #_w1);
   IF #_w1 THEN
       "SolutieB_DB"(esd := "Avarii".ESD,   // "Solutie"
                     avarie := "Avarii".avarie_generala,
                     debit_solutie := "Solutie_B_DB".debit_solutie,
                     debit_cerut := "Solutie_B_DB".debit_de_umplut,
                     resetare_sistem := "Simulare_DB".resetare_proces,
                     debit_aux := "Solutie_B_DB".debit_aux,
                     btn_reumplere_solutie := "Solutie_B_DB".btn_reumplere,
                     capacitate_necesara := "Solutie_B_DB".capacitate_necesara,
                     btn_pornire := "Solutie_B_DB".btn_pornire,
                     terminat_umplere := "Butoane/Permisiuni".terminat_umplere_B,
                     debit_curent => "Solutie_B_DB".debit_curent,
                     alarma => "Alarme".alarme_vect[6],
                     pornire_golire => "Solutie_B_DB".pornite_golire);
   END_IF;
END_REGION

REGION Network 11: Conditie de pornire
   RUNG wire#powerrail
      I_Contact( "Avarii".ESD )
      I_Contact( "Avarii".avarie_generala )
      Contact( "Butoane/Permisiuni".btn_start )
      I_Contact( "Auxiliare".intrece_limita_container )
      { S7_Templates := "SrcType := Time" } NE_Contact(in1 := "Mixer_DB".durata_mixer, in2 := T#0MS)
      { S7_Templates := "SrcType := UInt" } NE_Contact(in1 := "Container_DB".debit_total, in2 := 0)
      { S7_Templates := "SrcType := UInt" } NE_Contact(in1 := "Container_DB".debit_recipient, in2 := 0)
      { S7_Templates := "SrcType := UInt" } NE_Contact(in1 := "Solutie_A_DB".debit_solutie, in2 := 0)
      { S7_Templates := "SrcType := UInt" } NE_Contact(in1 := "Solutie_A_DB".debit_de_umplut, in2 := 0)
      { S7_Templates := "SrcType := UInt" } NE_Contact(in1 := "Solutie_B_DB".debit_solutie, in2 := 0)
      { S7_Templates := "SrcType := UInt" } NE_Contact(in1 := "Solutie_B_DB".debit_de_umplut, in2 := 0)
      Coil( "Butoane/Permisiuni".permisiune_start )
   END_RUNG
   // the same network as SCL:
   "Butoane/Permisiuni".permisiune_start := NOT "Avarii".ESD AND NOT "Avarii".avarie_generala AND "Butoane/Permisiuni".btn_start AND NOT "Auxiliare".intrece_limita_container AND ("Mixer_DB".durata_mixer <> T#0MS) AND ("Container_DB".debit_total <> 0) AND ("Container_DB".debit_recipient <> 0) AND ("Solutie_A_DB".debit_solutie <> 0) AND ("Solutie_A_DB".debit_de_umplut <> 0) AND ("Solutie_B_DB".debit_solutie <> 0) AND ("Solutie_B_DB".debit_de_umplut <> 0);
END_REGION

REGION Network 12: Verificare daca intrece limita containterului
   RUNG wire#powerrail
      Add(in1 := "Solutie_A_DB".debit_de_umplut, in2 := "Solutie_B_DB".debit_de_umplut, out => "Auxiliare".debit_suma)
      { S7_Templates := "SrcType := UInt" } GT_Contact(in1 := "Auxiliare".debit_suma, in2 := "Container_DB".debit_total)
      Coil( "Alarme".alarme_vect[7] )
      Coil( "Auxiliare".intrece_limita_container )
   END_RUNG
   // the same network as SCL:
   "Auxiliare".debit_suma := "Solutie_A_DB".debit_de_umplut + "Solutie_B_DB".debit_de_umplut;
   "Alarme".alarme_vect[7] := "Auxiliare".debit_suma > "Container_DB".debit_total;
   "Auxiliare".intrece_limita_container := "Auxiliare".debit_suma > "Container_DB".debit_total;
END_REGION

REGION Network 13: Simulare
   RUNG wire#powerrail
      "Simulare_DB_1"(permisiune_pornire := "Butoane/Permisiuni".permisiune_start, debit_A := "Solutie_A_DB".debit_aux, debit_B := "Solutie_B_DB".debit_aux, debit_cerut_total := "Auxiliare".debit_suma, terminat_A := "Butoane/Permisiuni".terminat_umplere_A, terminat_B := "Butoane/Permisiuni".terminat_umplere_B, terminat_mixer := "Butoane/Permisiuni".terminat_mixer, alarma_A := "Alarme".alarme_vect[5], alarma_B := "Alarme".alarme_vect[6], terminat_golire := "Butoane/Permisiuni".terminat_golire, debit_container := "Container_DB".debit_curent, plecare_A := "Solutie_A_DB".btn_pornire, plecare_B := "Solutie_B_DB".btn_pornire, resetare_proces := "Simulare_DB".resetare_proces, pornire_mixer => "Mixer_DB".btn_pornire, pornire_golire => "Container_DB".btn_pornire, terminat_umplere => "Butoane/Permisiuni".terminat_umplere, terminat_proces => "Simulare_DB".terminat_proces, alarma_terminat => "Alarme".alarme_vect[8])
   END_RUNG
   // the same network as SCL:
   "Simulare_DB_1"(permisiune_pornire := "Butoane/Permisiuni".permisiune_start,   // "Simulare"
                   debit_A := "Solutie_A_DB".debit_aux,
                   debit_B := "Solutie_B_DB".debit_aux,
                   debit_cerut_total := "Auxiliare".debit_suma,
                   terminat_A := "Butoane/Permisiuni".terminat_umplere_A,
                   terminat_B := "Butoane/Permisiuni".terminat_umplere_B,
                   terminat_mixer := "Butoane/Permisiuni".terminat_mixer,
                   alarma_A := "Alarme".alarme_vect[5],
                   alarma_B := "Alarme".alarme_vect[6],
                   terminat_golire := "Butoane/Permisiuni".terminat_golire,
                   debit_container := "Container_DB".debit_curent,
                   plecare_A := "Solutie_A_DB".btn_pornire,
                   plecare_B := "Solutie_B_DB".btn_pornire,
                   resetare_proces := "Simulare_DB".resetare_proces,
                   pornire_mixer => "Mixer_DB".btn_pornire,
                   pornire_golire => "Container_DB".btn_pornire,
                   terminat_umplere => "Butoane/Permisiuni".terminat_umplere,
                   terminat_proces => "Simulare_DB".terminat_proces,
                   alarma_terminat => "Alarme".alarme_vect[8]);
END_REGION

REGION Network 14: Reseteaza butonul de start daca s-a terminat
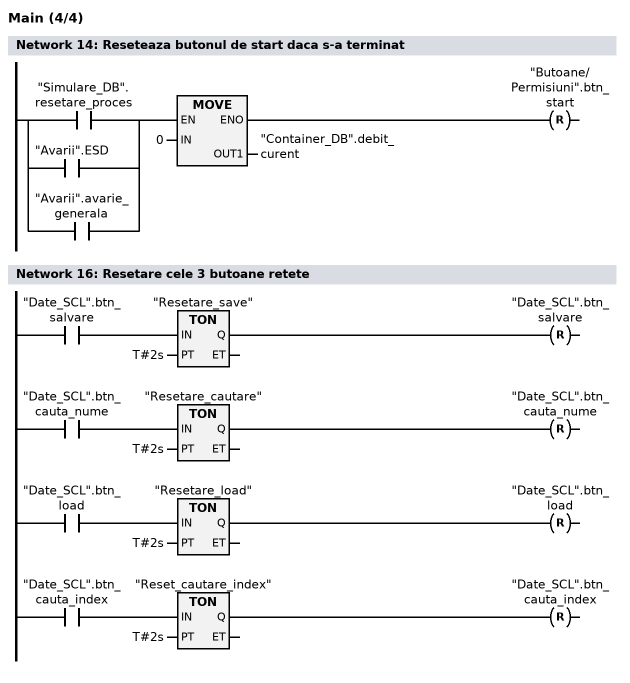
   RUNG wire#powerrail
      Contact( "Simulare_DB".resetare_proces )
      wire#w1
      Move(in := 0, out1 => "Container_DB".debit_curent)
      R_Coil( "Butoane/Permisiuni".btn_start )
   END_RUNG
   RUNG wire#powerrail
      Contact( "Avarii".ESD )
   END_RUNG wire#w1
   RUNG wire#powerrail
      Contact( "Avarii".avarie_generala )
   END_RUNG wire#w1
   // the same network as SCL:
   IF "Simulare_DB".resetare_proces OR "Avarii".ESD OR "Avarii".avarie_generala THEN
       "Container_DB".debit_curent := 0;
       "Butoane/Permisiuni".btn_start := FALSE;
   END_IF;
END_REGION

REGION Network 15 (SCL): Retete pt HMI (reteta proprie a la chef Scarlatescu)
   IF "Date_SCL".index > 99 OR "Date_SCL".index < 0 THEN//v1, just left it in case of anything
       "Alarme".alarme_vect[9] := TRUE;
       //RETURN;
   ELSIF "Date_SCL".valoare_cantitate_A > 60 OR "Date_SCL".valoare_cantitate_B > 60 THEN
       "Alarme".alarme_vect[11] := TRUE;
       //RETURN;
   ELSIF "Date_SCL".valoare_cantitate_A <= 60 OR "Date_SCL".valoare_cantitate_B <= 60 THEN
       "Alarme".alarme_vect[11] := FALSE;
       //RETURN;
       IF "Date_SCL".btn_cauta_nume THEN
           IF "Date_SCL".nume = '' THEN
               "Alarme".alarme_vect[12] := TRUE;
               RETURN;
           ELSE
               "Alarme".alarme_vect[12] := FALSE;
               FOR "Date_SCL".index_for := 0 TO 99 DO
                   IF "Date_SCL".array_nume["Date_SCL".index_for] = "Date_SCL".nume THEN
                       "Date_SCL".index := "Date_SCL".index_for;
                       "Alarme".alarme_vect[13] := FALSE;
                       EXIT;
                   ELSE
                       "Alarme".alarme_vect[13] := TRUE;
                   END_IF;
               END_FOR;
               IF "Alarme".alarme_vect[13] = FALSE THEN
                   "Date_SCL".valoare_durata := "Date_SCL".array_durata["Date_SCL".index];
                   "Date_SCL".valoare_cantitate_A := "Date_SCL".array_cantitate_A["Date_SCL".index];
                   "Date_SCL".valoare_cantitate_B := "Date_SCL".array_cantitate_B["Date_SCL".index];
                   "Date_SCL".nume := "Date_SCL".array_nume["Date_SCL".index];
               END_IF;
           END_IF;
       ELSIF "Date_SCL".btn_cauta_index THEN
           "Date_SCL".valoare_durata := "Date_SCL".array_durata["Date_SCL".index];
           "Date_SCL".valoare_cantitate_A := "Date_SCL".array_cantitate_A["Date_SCL".index];
           "Date_SCL".valoare_cantitate_B := "Date_SCL".array_cantitate_B["Date_SCL".index];
           "Date_SCL".nume := "Date_SCL".array_nume["Date_SCL".index];
       ELSIF "Date_SCL".btn_salvare THEN
           IF "Date_SCL".valoare_cantitate_A = 0 OR "Date_SCL".valoare_cantitate_B = 0 OR "Date_SCL".valoare_durata = T#0ms OR "Date_SCL".nume = '' THEN
               "Alarme".alarme_vect[10] := TRUE;
               //RETURN;
           ELSE
               "Date_SCL".array_cantitate_A["Date_SCL".index] := "Date_SCL".valoare_cantitate_A;
               "Date_SCL".array_cantitate_B["Date_SCL".index] := "Date_SCL".valoare_cantitate_B;
               "Date_SCL".array_durata["Date_SCL".index] := "Date_SCL".valoare_durata;
               "Date_SCL".array_nume["Date_SCL".index] := "Date_SCL".nume;
               "Alarme".alarme_vect[10] := FALSE;
           END_IF;
       ELSIF "Date_SCL".btn_load THEN
           IF "Date_SCL".valoare_cantitate_A = 0 OR "Date_SCL".valoare_cantitate_B = 0 OR "Date_SCL".valoare_durata = T#0ms OR "Date_SCL".nume = '' THEN
               "Alarme".alarme_vect[10] := TRUE;
               //RETURN;
           ELSE
               "Mixer_DB".durata_mixer := "Date_SCL".valoare_durata;
               "Solutie_A_DB".debit_de_umplut := "Date_SCL".valoare_cantitate_A;
               "Solutie_B_DB".debit_de_umplut := "Date_SCL".valoare_cantitate_B;
               "Simulare_DB".nume := "Date_SCL".nume;
               "Alarme".alarme_vect[10] := FALSE;
           END_IF;
       END_IF;
       ELSE
           RETURN;
   END_IF;
END_REGION

REGION Network 16: Resetare cele 3 butoane retete
   "Resetare_save".TON(IN := "Date_SCL".btn_salvare, PT := T#2s);
   IF "Resetare_save".Q THEN "Date_SCL".btn_salvare := FALSE; END_IF;
   "Resetare_cautare".TON(IN := "Date_SCL".btn_cauta_nume, PT := T#2s);
   IF "Resetare_cautare".Q THEN "Date_SCL".btn_cauta_nume := FALSE; END_IF;
   "Resetare_load".TON(IN := "Date_SCL".btn_load, PT := T#2s);
   IF "Resetare_load".Q THEN "Date_SCL".btn_load := FALSE; END_IF;
   "Reset_cautare_index".TON(IN := "Date_SCL".btn_cauta_index, PT := T#2s);
   IF "Reset_cautare_index".Q THEN "Date_SCL".btn_cauta_index := FALSE; END_IF;
END_REGION
END_ORGANIZATION_BLOCK

(* ===== HMI "HMI_RT_1" =====
system functions are stored by id; their names below are inferred from use
connection "HMI_Connection_1": ETHERNET, SMART_S7_1500_OMS

HMI tags "Default tag table"
   "Tag_ScreenNumber" : UInt, internal
   "Alarme_alarme_gather" : Word = PLC Alarme.alarme_gather, 1 s
   "Avarii_ESD" : Bool = PLC Avarii.ESD, 1 s
   "Avarii_avarie_mixer" : Bool = PLC Avarii.avarie_mixer, 1 s
   "Avarii_avarie_container" : Bool = PLC Avarii.avarie_container, 1 s
   "Avarii_avarie_solutie_A" : Bool = PLC Avarii.avarie_solutie_A, 1 s
   "Avarii_avarie_solutie_B" : Bool = PLC Avarii.avarie_solutie_B, 1 s
   "Avarii_reset_avarie_generala" : Bool = PLC Avarii.reset_avarie_generala, 1 s
   "Avarii_avarie_generala" : Bool = PLC Avarii.avarie_generala, 1 s
   "Avarii_reset_esd" : Bool = PLC Avarii.reset_esd, 1 s
   "Avarii_esd_btn" : Bool = PLC Avarii.esd_btn, 1 s
   "Mixer_DB_durata_mixer" : Time = PLC Mixer_DB.durata_mixer, 1 s
   "Solutie_A_DB_debit_de_umplut" : UInt = PLC Solutie_A_DB.debit_de_umplut, 1 s
   "Solutie_B_DB_debit_de_umplut" : UInt = PLC Solutie_B_DB.debit_de_umplut, 1 s
   "Solutie_B_DB_debit_curent" : UInt = PLC Solutie_B_DB.debit_curent, 1 s
   "Butoane/Permisiuni_btn_start" : Bool = PLC "Butoane/Permisiuni".btn_start, 1 s
   "Solutie_A_DB_debit_curent" : UInt = PLC Solutie_A_DB.debit_curent, 1 s
   "Solutie_A_DB_btn_reumplere" : Bool = PLC Solutie_A_DB.btn_reumplere, 1 s
   "Container_DB_debit_curent" : UInt = PLC Container_DB.debit_curent, 1 s
   "Container_DB_debit_total" : UInt = PLC Container_DB.debit_total, 1 s
   "Container_DB_recipient" : Bool = PLC Container_DB.recipient, 1 s
   "Container_DB_valva_golire_deschisa" : Bool = PLC Container_DB.valva_golire_deschisa, 1 s
   "Solutie_A_DB_pornite_golire" : Bool = PLC Solutie_A_DB.pornite_golire, 1 s
   "Solutie_B_DB_pornite_golire" : Bool = PLC Solutie_B_DB.pornite_golire, 1 s
   "Mixer_DB_mixer_pornit" : Bool = PLC Mixer_DB.mixer_pornit, 1 s
   "Simulare_DB_resetare_proces" : Bool = PLC Simulare_DB.resetare_proces, 1 s
   "Solutie_B_DB_btn_reumplere" : Bool = PLC Solutie_B_DB.btn_reumplere, 1 s
   "Mixer_DB_timp_elapsed" : Time = PLC Mixer_DB.timp_elapsed, 1 s
   "Variabile_HMI_stea_1" : Bool = PLC Variabile_HMI.stea_1, 1 s
   "Variabile_HMI_stea_2" : Bool = PLC Variabile_HMI.stea_2, 1 s
   "Variabile_HMI_triunghi_1" : Bool = PLC Variabile_HMI.triunghi_1, 1 s
   "Variabile_HMI_triunghi_2" : Bool = PLC Variabile_HMI.triunghi_2, 1 s
   "Date_SCL_index" : Int = PLC Date_SCL.index, 1 s
   "Date_SCL_valoare_durata" : Time = PLC Date_SCL.valoare_durata, 1 s
   "Date_SCL_valoare_cantitate_B" : UInt = PLC Date_SCL.valoare_cantitate_B, 1 s
   "Date_SCL_valoare_cantitate_A" : UInt = PLC Date_SCL.valoare_cantitate_A, 1 s
   "Date_SCL_btn_salvare" : Bool = PLC Date_SCL.btn_salvare, 1 s
   "Date_SCL_btn_cauta_nume" : Bool = PLC Date_SCL.btn_cauta_nume, 1 s
   "Date_SCL_btn_load" : Bool = PLC Date_SCL.btn_load, 1 s
   "Auxiliare_debit_suma" : UInt = PLC Auxiliare.debit_suma, 1 s
   "Date_SCL_nume" : String[254] = PLC Date_SCL.nume, 1 s
   "Simulare_DB_nume" : String[254] = PLC Simulare_DB.nume, 1 s
   "Date_SCL_btn_cauta_index" : Bool = PLC Date_SCL.btn_cauta_index, 1 s

discrete alarms
   1: 'ESD', class Errors, trigger "Alarme_alarme_gather" bit 0
   2: 'Avarie mixer', class Errors, trigger "Alarme_alarme_gather" bit 1
   3: 'Avarie container', class Errors, trigger "Alarme_alarme_gather" bit 2
   4: 'Avarie solutie A', class Errors, trigger "Alarme_alarme_gather" bit 3
   5: 'Avarie solutie B', class Errors, trigger "Alarme_alarme_gather" bit 4
   6: 'A nu are suficienta solutie', class Errors, trigger "Alarme_alarme_gather" bit 5
   7: 'B nu are suficienta solutie', class Errors, trigger "Alarme_alarme_gather" bit 6
   8: 'Limita depasita (A + B > limita container)', class Errors, trigger "Alarme_alarme_gather" bit 7
   9: 'Proces terminat, resetati sistemul', class Errors, trigger "Alarme_alarme_gather" bit 8
   10: 'Index out of bounds la retete', class Errors, trigger "Alarme_alarme_gather" bit 9
   11: 'Reteta este incompleta (una din valori este 0)', class Errors, trigger "Alarme_alarme_gather" bit 10
   12: 'Cerere peste volumul maxim de solutie', class Errors, trigger "Alarme_alarme_gather" bit 11
   13: 'Numele este gol, nu poate fi cautat', class Errors, trigger "Alarme_alarme_gather" bit 12
   14: 'Numele nu a fost gasit in DB', class Errors, trigger "Alarme_alarme_gather" bit 13

recipe "Vopsea": Durata <- "Mixer_DB_durata_mixer", Cantitate_A <- "Solutie_A_DB_debit_de_umplut", Cantitate_B <- "Solutie_B_DB_debit_de_umplut"

recipe "Chimicale": Durata <- "Mixer_DB_durata_mixer", Cantitate_A <- "Solutie_A_DB_debit_de_umplut", Cantitate_B <- "Solutie_B_DB_debit_de_umplut"

screen "Simulare" 800x480, template "Template_1"
   on GenerateScreen: SetTag("Tag_ScreenNumber", 1)
   TextField "Text field_1" at 23,445 size 60x20; Text 'Simulare'
   TextField "Text field_2" at 131,444 size 43x20; Text 'Avarii'
   TextField "Text field_3" at 226,443 size 50x20; Text 'Retete'
   Button "Button_1" at 37,69 size 58x32; TextOff 'ESD'
   Button "Button_2" at 37,110 size 59x32; TextOff 'Reset'
   TextField "Text field_4" at 362,18 size 97x29; Text 'Simulare'
   Rectangle "Rectangle_4" at 545,236 size 49x15
      Appearance <- "Solutie_B_DB_pornite_golire"
   Rectangle "Rectangle_5" at 340,236 size 49x15
      Appearance <- "Solutie_A_DB_pornite_golire"
   Rectangle "Rectangle_6" at 456,383 size 23x21
      Appearance <- "Container_DB_valva_golire_deschisa"
   Rectangle "Rectangle_7" at 419,413 size 96x48
      Appearance <- "Container_DB_recipient"
   Bar "Bar_1" at 394,203 size 145x173; MinimumValue 0; MaximumValue 100
      ProcessValue <- "Container_DB_debit_curent"
   Bar "Bar_2" at 600,146 size 104x105; MinimumValue 0; MaximumValue 60
      ProcessValue <- "Solutie_B_DB_debit_curent"
   Bar "Bar_3" at 230,147 size 104x105; MinimumValue 0; MaximumValue 60
      ProcessValue <- "Solutie_A_DB_debit_curent"
   IOField "I/O field_1" at 554,334 size 58x32; FormatPattern 999; Unit L
      ProcessValue <- "Container_DB_debit_curent"
   TextField "Text field_5" at 557,309 size 49x20; Text 'Curent'
   IOField "I/O field_2" at 251,101 size 58x32; FormatPattern 999; Unit L
      ProcessValue <- "Solutie_A_DB_debit_curent"
   TextField "Text field_6" at 254,76 size 49x20; Text 'Curent'
   IOField "I/O field_3" at 625,101 size 58x32; FormatPattern 999; Unit L
      ProcessValue <- "Solutie_B_DB_debit_curent"
   TextField "Text field_7" at 628,76 size 49x20; Text 'Curent'
   Button "Button_3" at 628,269 size 60x32; TextOff 'Umplere'
      on Click: SetBit("Solutie_B_DB_btn_reumplere")
   Button "Button_4" at 255,269 size 60x32; TextOff 'Umplere'
      on Activate: SetBit("Solutie_A_DB_btn_reumplere")
   GraphicView "Graphic view_2" at 426,57 size 83x238; Picture "Graphic_2"
      Visibility <- "Mixer_DB_mixer_pornit"
   GraphicView "Graphic view_1" at 427,57 size 83x238; Picture "Graphic_1"
      Visibility <- "Avarii_avarie_mixer"
   GraphicView "Graphic view_3" at 427,57 size 83x238; Picture "Graphic_3"
      Visibility <- "Variabile_HMI_triunghi_2"
   GraphicView "Graphic view_4" at 427,57 size 83x238; Picture "Graphic_4"
      Visibility <- "Variabile_HMI_triunghi_1"
   GraphicView "Graphic view_6" at 427,57 size 83x238; Picture "Graphic_6"
      Visibility <- "Variabile_HMI_stea_1"
   GraphicView "Graphic view_5" at 427,57 size 83x238; Picture "Graphic_5"
      Visibility <- "Variabile_HMI_stea_2"
   IOField "I/O field_4" at 322,333 size 58x32; FormatPattern 999; Unit L
      ProcessValue <- "Container_DB_debit_total"
   TextField "Text field_8" at 331,308 size 37x20; Text 'Total'
   Button "Button_5" at 68,257 size 96x32; TextOff 'Start'
      on Click: SetBit("Butoane/Permisiuni_btn_start")
   TextField "Text field_9" at 271,51 size 17x25; Text 'A'
   TextField "Text field_10" at 643,51 size 17x25; Text 'B'
   Button "Button_6" at 68,300 size 96x32; TextOff 'Reset'
      on Click: SetBit("Simulare_DB_resetare_proces")
   Button "Button_7" at 532,420 size 68x32; TextOff 'Recipient'
      on Click: SetBit("Container_DB_recipient")
   IOField "I/O field_5" at 529,37 size 50x32; FormatPattern 999; Unit s
      ProcessValue <- "Mixer_DB_timp_elapsed"
   IOField "I/O field_6" at 262,304 size 47x32; FormatPattern 999; Unit L
      ProcessValue <- "Solutie_A_DB_debit_de_umplut"
   IOField "I/O field_7" at 635,304 size 45x32; FormatPattern 999; Unit L
      ProcessValue <- "Solutie_B_DB_debit_de_umplut"
   IOField "I/O field_8" at 135,15 size 114x32; FormatPattern ????????????????????????????????????????????????????????????????????????????????
      ProcessValue <- "Simulare_DB_nume"

screen "Retete" 800x480
   TextField "Text field_1" at 23,445 size 60x20; Text 'Simulare'
   TextField "Text field_2" at 131,444 size 43x20; Text 'Avarii'
   TextField "Text field_3" at 226,443 size 50x20; Text 'Retete'
   TextField "Text field_4" at 370,18 size 74x29; Text 'Retete'
   IOField "I/O field_1" at 201,90 size 96x32; FormatPattern ????????????????????
      ProcessValue <- "Date_SCL_nume"
   IOField "I/O field_2" at 202,205 size 96x32; FormatPattern 999; Unit s
      ProcessValue <- "Date_SCL_valoare_durata"
   IOField "I/O field_3" at 201,266 size 96x32; FormatPattern 999; Unit L
      ProcessValue <- "Date_SCL_valoare_cantitate_A"
   IOField "I/O field_4" at 202,327 size 96x32; FormatPattern 999; Unit L
      ProcessValue <- "Date_SCL_valoare_cantitate_B"
   TextField "Text field_5" at 137,92 size 40x20; Text 'Nume'
   TextField "Text field_6" at 131,205 size 50x20; Text 'Durata'
   TextField "Text field_7" at 131,272 size 53x20; Text 'Cant. A'
   TextField "Text field_8" at 132,333 size 51x20; Text 'Cant. B'
   Button "Button_1" at 496,121 size 96x32; TextOff 'Save'
      on Click: SetBit("Date_SCL_btn_salvare")
   Button "Button_2" at 496,180 size 96x32; TextOff 'Cauta nume'
      on Click: SetBit("Date_SCL_btn_cauta_nume")
   Button "Button_3" at 496,301 size 96x32; TextOff 'Load'
      on Click: SetBit("Date_SCL_btn_load")
   IOField "I/O field_5" at 202,144 size 96x32; FormatPattern 99
      ProcessValue <- "Date_SCL_index"
   TextField "Text field_9" at 138,146 size 41x20; Text 'Index'
   Button "Button_4" at 496,240 size 96x32; TextOff 'Cauta index'
      on Click: SetBit("Date_SCL_btn_cauta_index")

screen "Avarii" 800x480
   TextField "Text field_1" at 23,445 size 60x20; Text 'Simulare'
   TextField "Text field_2" at 131,444 size 43x20; Text 'Avarii'
   TextField "Text field_3" at 226,443 size 50x20; Text 'Retete'
   Button "Button_1" at 37,69 size 58x32; TextOff 'ESD'
      on Click: SetBit("Avarii_esd_btn")
   Button "Button_2" at 37,110 size 59x32; TextOff 'Reset'
      on Click: SetBit("Avarii_reset_esd")
   Circle "Circle_1" at 46,18 size 39x39
      Appearance <- "Avarii_ESD"
   TextField "Text field_4" at 370,18 size 65x29; Text 'Avarii'
   Circle "Circle_2" at 584,155 size 42x42
      Appearance <- "Avarii_avarie_mixer"
   Button "Button_3" at 658,160 size 96x32; TextOff 'Mixer'
      on Click: SetBit("Avarii_avarie_mixer")
   Circle "Circle_3" at 584,218 size 42x42
      Appearance <- "Avarii_avarie_container"
   Button "Button_4" at 658,223 size 96x32; TextOff 'Container'
      on Click: SetBit("Avarii_avarie_container")
   Circle "Circle_4" at 585,281 size 42x42
      Appearance <- "Avarii_avarie_solutie_A"
   Button "Button_5" at 659,286 size 96x32; TextOff 'Subst. A'
      on Click: SetBit("Avarii_avarie_solutie_A")
   Circle "Circle_5" at 585,343 size 42x42
      Appearance <- "Avarii_avarie_solutie_B"
   Button "Button_6" at 659,348 size 96x32; TextOff 'Subst. B'
      on Click: SetBit("Avarii_avarie_solutie_B")
   Button "Button_7" at 624,410 size 96x32; TextOff 'Reset'
      on Click: SetBit("Avarii_reset_avarie_generala")
   Circle "Circle_6" at 644,51 size 63x63
      Appearance <- "Avarii_avarie_generala"
   TextField "Text field_5" at 612,21 size 124x22; Text 'Avarie generala'
*)